FUNCTION_BLOCK AUS_TO_ADI (* Composite FB for converting AUS (USINT) adapter to ADI (DINT) adapter *)
  (* Standard: 61499-2; Description: Copyright (c) 2026 HR Agrartechnik GmbH This program and the accompanying materials are made available under the terms of the Eclipse Public License 2.0 which is available at https://www.eclipse.org/legal/epl-2.0/ SPDX-License-Identifier: EPL-2.0 *)
  (* Version 1.0, 2026-02-17, Franz Höpfinger, HR Agrartechnik GmbH *)
  PACKAGE adapter::conversion::unidirectional;
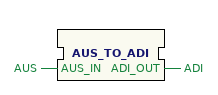
  SOCKETS
    AUS_IN : adapter::types::unidirectional::AUS; (* USINT Adapter Input *)
  END_SOCKETS
  PLUGS
    ADI_OUT : adapter::types::unidirectional::ADI; (* DINT Adapter Output *)
  END_PLUGS
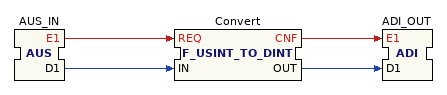
  FBS
    Convert : iec61131::conversion::F_USINT_TO_DINT;
  END_FBS
  EVENT_CONNECTIONS
    AUS_IN.E1 TO Convert.REQ;
    Convert.CNF TO ADI_OUT.E1;
  END_CONNECTIONS
  DATA_CONNECTIONS
    AUS_IN.D1 TO Convert.IN;
    Convert.OUT TO ADI_OUT.D1;
  END_CONNECTIONS
END_FUNCTION_BLOCK
